# EPICS substitutions: db/ecmcEK1101.substitutions
file ecmcEcSlave.template
{
    pattern {}
            {}
}

file ecmcEK1101.template
{
	pattern {}
		    {}
}
